// TIA Portal V16 export
// export: Created 2025-12-18T09:29:14.422134Z, ExportSetting WithDefaults, DisplayName Totally Integrated Automation Portal, DisplayVersion V16, DisplayName TIA Portal Version Control Interface, DisplayVersion V16, DisplayName TIA Portal Openness, DisplayVersion V16, DisplayName STEP 7 Professional, DisplayVersion V16, DisplayName STEP 7 Safety, DisplayVersion V16, DisplayName WinCC Advanced, DisplayVersion V16
FUNCTION_BLOCK "Work Station"   // FB1, LAD
{ S7_Optimized_Access := 'TRUE' }
VERSION : 0.1
// stored: AutoNumber true, IsIECCheckEnabled false, IsRetainMemResEnabled false, MemoryReserve 100, SetENOAutomatically false, UDAEnableTagReadback false
   VAR_INPUT
      xEntrySensor { ExternalAccessible := 'False'; ExternalVisible := 'False'; ExternalWritable := 'False'} : Bool;
      xExitSensor { ExternalAccessible := 'False'; ExternalVisible := 'False'; ExternalWritable := 'False'} : Bool;
      xPositionerSensor { ExternalAccessible := 'False'; ExternalVisible := 'False'; ExternalWritable := 'False'} : Bool;
      xQueueSensor { ExternalAccessible := 'False'; ExternalVisible := 'False'; ExternalWritable := 'False'} : Bool;
      xClampSensor { ExternalAccessible := 'False'; ExternalVisible := 'False'; ExternalWritable := 'False'} : Bool;
   END_VAR
   VAR_IN_OUT
      xConveyor1 { ExternalAccessible := 'False'; ExternalVisible := 'False'; ExternalWritable := 'False'} : Bool;
      xConveyor2 { ExternalAccessible := 'False'; ExternalVisible := 'False'; ExternalWritable := 'False'} : Bool;
      xConveyor3 { ExternalAccessible := 'False'; ExternalVisible := 'False'; ExternalWritable := 'False'} : Bool;
      xPositionerClamp : Bool;
      xPositionerRaise : Bool;
      "Work Station DB" : "UDT WorkStation";
   END_VAR
   VAR
      StationConveyorControl_Instance { S7_SetPoint := 'True'} : "StationConveyorControl";
      StationProcessControl_Instance { S7_SetPoint := 'True'} : "StationProcessControl";
   END_VAR
BEGIN

REGION Network 2
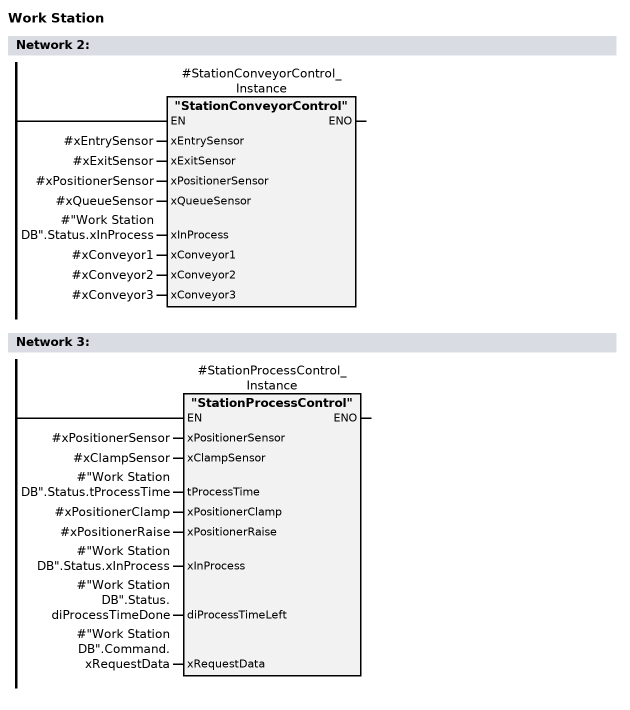
   RUNG wire#powerrail
      #StationConveyorControl_Instance(xEntrySensor := #xEntrySensor, xExitSensor := #xExitSensor, xPositionerSensor := #xPositionerSensor, xQueueSensor := #xQueueSensor, xInProcess := #"Work Station DB".Status.xInProcess, xConveyor1 := #xConveyor1, xConveyor2 := #xConveyor2, xConveyor3 := #xConveyor3)
   END_RUNG
   // the same network as SCL:
   #StationConveyorControl_Instance(xEntrySensor := #xEntrySensor,   // "StationConveyorControl"
                           xExitSensor := #xExitSensor,
                           xPositionerSensor := #xPositionerSensor,
                           xQueueSensor := #xQueueSensor,
                           xInProcess := #"Work Station DB".Status.xInProcess,
                           xConveyor1 := #xConveyor1,
                           xConveyor2 := #xConveyor2,
                           xConveyor3 := #xConveyor3);
END_REGION

REGION Network 3
   RUNG wire#powerrail
      #StationProcessControl_Instance(xPositionerSensor := #xPositionerSensor, xClampSensor := #xClampSensor, tProcessTime := #"Work Station DB".Status.tProcessTime, xPositionerClamp := #xPositionerClamp, xPositionerRaise := #xPositionerRaise, xInProcess := #"Work Station DB".Status.xInProcess, diProcessTimeLeft := #"Work Station DB".Status.diProcessTimeDone, xRequestData := #"Work Station DB".Command.xRequestData)
   END_RUNG
   // the same network as SCL:
   #StationProcessControl_Instance(xPositionerSensor := #xPositionerSensor,   // "StationProcessControl"
                           xClampSensor := #xClampSensor,
                           tProcessTime := #"Work Station DB".Status.tProcessTime,
                           xPositionerClamp := #xPositionerClamp,
                           xPositionerRaise := #xPositionerRaise,
                           xInProcess := #"Work Station DB".Status.xInProcess,
                           diProcessTimeLeft := #"Work Station DB".Status.diProcessTimeDone,
                           xRequestData := #"Work Station DB".Command.xRequestData);
END_REGION
END_FUNCTION_BLOCK
